TYPE EL1852_Data :
STRUCT
	{attribute addProperty Name "1"}
	{attribute addProperty Name "Channel 1"}
	_1 :DiChannel;
	{attribute addProperty Name "Channel 2"}
	_2 :DiChannel;
	{attribute addProperty Name "Channel 3"}
	_3 :DiChannel;
	{attribute addProperty Name "Channel 4"}
	_4 :DiChannel;
	{attribute addProperty Name "Channel 5"}
	_5 :DiChannel;
	{attribute addProperty Name "Channel 6"}
	_6 :DiChannel;
	{attribute addProperty Name "Channel 7"}
	_7 :DiChannel;
	{attribute addProperty Name "Channel 8"}
	_8 :DiChannel;
	{attribute addProperty Name "Channel 9"}
	_9 :DoChannel;
	{attribute addProperty Name "Channel 10"}
	_10 :DoChannel;
	{attribute addProperty Name "Channel 11"}
	_11 :DoChannel;
	{attribute addProperty Name "Channel 12"}
	_12 :DoChannel;
	{attribute addProperty Name "Channel 13"}
	_13 :DoChannel;
	{attribute addProperty Name "Channel 14"}
	_14 :DoChannel;
	{attribute addProperty Name "Channel 15"}
	_15 :DoChannel;
	{attribute addProperty Name "Channel 16"}
	_16 :DoChannel;
END_STRUCT
END_TYPE

(* stored: Version 1.1.0.1, ProductVersion 3.1.4024.9
   DUT EL1852_Data: Id {56cb11ef-a201-0115-3116-be1b687102d0} *)
